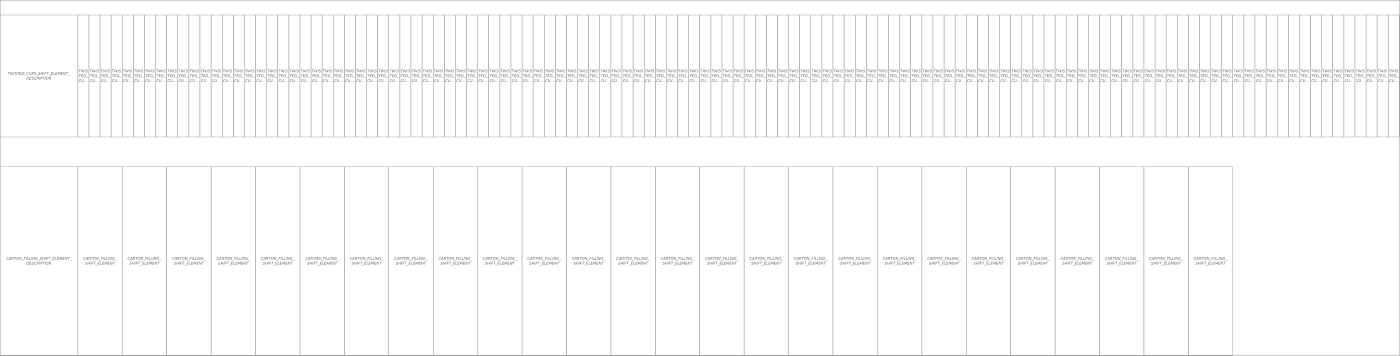
VISUALIZATION CUPS_PICK_AND_PLACE  // 3782x962
    Frame (210,40 30x330)
        shows TWISTED_CUPS_SHIFT_ELEMENT(index := 50)
    Frame (240,40 30x330)
        shows TWISTED_CUPS_SHIFT_ELEMENT(index := 51)
    Frame (270,40 30x330)
        shows TWISTED_CUPS_SHIFT_ELEMENT(index := 52)
    Frame (300,40 30x330)
        shows TWISTED_CUPS_SHIFT_ELEMENT(index := 53)
    Frame (330,40 30x330)
        shows TWISTED_CUPS_SHIFT_ELEMENT(index := 54)
    Frame (360,40 30x330)
        shows TWISTED_CUPS_SHIFT_ELEMENT(index := 55)
    Frame (390,40 30x330)
        shows TWISTED_CUPS_SHIFT_ELEMENT(index := 56)
    Frame (420,40 30x330)
        shows TWISTED_CUPS_SHIFT_ELEMENT(index := 57)
    Frame (450,40 30x330)
        shows TWISTED_CUPS_SHIFT_ELEMENT(index := 58)
    Frame (480,40 30x330)
        shows TWISTED_CUPS_SHIFT_ELEMENT(index := 59)
    Frame (510,40 30x330)
        shows TWISTED_CUPS_SHIFT_ELEMENT(index := 60)
    Frame (0,40 210x330)
        shows TWISTED_CUPS_SHIFT_ELEMENT_DESCRIPTION()
    Frame (540,40 30x330)
        shows TWISTED_CUPS_SHIFT_ELEMENT(index := 61)
    Frame (570,40 30x330)
        shows TWISTED_CUPS_SHIFT_ELEMENT(index := 62)
    Frame (600,40 30x330)
        shows TWISTED_CUPS_SHIFT_ELEMENT(index := 63)
    Frame (630,40 30x330)
        shows TWISTED_CUPS_SHIFT_ELEMENT(index := 64)
    Frame (660,40 30x330)
        shows TWISTED_CUPS_SHIFT_ELEMENT(index := 65)
    Frame (690,40 30x330)
        shows TWISTED_CUPS_SHIFT_ELEMENT(index := 66)
    Frame (720,40 30x330)
        shows TWISTED_CUPS_SHIFT_ELEMENT(index := 67)
    Frame (750,40 30x330)
        shows TWISTED_CUPS_SHIFT_ELEMENT(index := 68)
    Frame (780,40 30x330)
        shows TWISTED_CUPS_SHIFT_ELEMENT(index := 69)
    Frame (810,40 30x330)
        shows TWISTED_CUPS_SHIFT_ELEMENT(index := 70)
    Frame (840,40 30x330)
        shows TWISTED_CUPS_SHIFT_ELEMENT(index := 71)
    Frame (870,40 30x330)
        shows TWISTED_CUPS_SHIFT_ELEMENT(index := 72)
    Frame (900,40 30x330)
        shows TWISTED_CUPS_SHIFT_ELEMENT(index := 73)
    Frame (930,40 30x330)
        shows TWISTED_CUPS_SHIFT_ELEMENT(index := 74)
    Frame (960,40 30x330)
        shows TWISTED_CUPS_SHIFT_ELEMENT(index := 75)
    Frame (990,40 30x330)
        shows TWISTED_CUPS_SHIFT_ELEMENT(index := 76)
    Frame (1020,40 30x330)
        shows TWISTED_CUPS_SHIFT_ELEMENT(index := 77)
    Frame (1050,40 30x330)
        shows TWISTED_CUPS_SHIFT_ELEMENT(index := 78)
    Frame (1080,40 30x330)
        shows TWISTED_CUPS_SHIFT_ELEMENT(index := 79)
    Frame (1110,40 30x330)
        shows TWISTED_CUPS_SHIFT_ELEMENT(index := 80)
    Frame (1140,40 30x330)
        shows TWISTED_CUPS_SHIFT_ELEMENT(index := 81)
    Frame (1170,40 30x330)
        shows TWISTED_CUPS_SHIFT_ELEMENT(index := 82)
    Frame (1200,40 30x330)
        shows TWISTED_CUPS_SHIFT_ELEMENT(index := 83)
    Frame (1230,40 30x330)
        shows TWISTED_CUPS_SHIFT_ELEMENT(index := 84)
    Frame (1260,40 30x330)
        shows TWISTED_CUPS_SHIFT_ELEMENT(index := 85)
    Frame (1290,40 30x330)
        shows TWISTED_CUPS_SHIFT_ELEMENT(index := 86)
    Frame (1320,40 30x330)
        shows TWISTED_CUPS_SHIFT_ELEMENT(index := 87)
    Frame (1350,40 30x330)
        shows TWISTED_CUPS_SHIFT_ELEMENT(index := 88)
    Frame (1380,40 30x330)
        shows TWISTED_CUPS_SHIFT_ELEMENT(index := 89)
    Frame (1410,40 30x330)
        shows TWISTED_CUPS_SHIFT_ELEMENT(index := 90)
    Frame (1440,40 30x330)
        shows TWISTED_CUPS_SHIFT_ELEMENT(index := 91)
    Frame (1470,40 30x330)
        shows TWISTED_CUPS_SHIFT_ELEMENT(index := 92)
    Frame (1500,40 30x330)
        shows TWISTED_CUPS_SHIFT_ELEMENT(index := 93)
    Frame (1530,40 30x330)
        shows TWISTED_CUPS_SHIFT_ELEMENT(index := 94)
    Frame (1560,40 30x330)
        shows TWISTED_CUPS_SHIFT_ELEMENT(index := 95)
    Frame (1590,40 30x330)
        shows TWISTED_CUPS_SHIFT_ELEMENT(index := 96)
    Frame (1620,40 30x330)
        shows TWISTED_CUPS_SHIFT_ELEMENT(index := 97)
    Frame (1650,40 30x330)
        shows TWISTED_CUPS_SHIFT_ELEMENT(index := 98)
    Frame (1680,40 30x330)
        shows TWISTED_CUPS_SHIFT_ELEMENT(index := 99)
    Frame (1710,40 30x330)
        shows TWISTED_CUPS_SHIFT_ELEMENT(index := 100)
    Frame (1740,40 30x330)
        shows TWISTED_CUPS_SHIFT_ELEMENT(index := 101)
    Frame (1770,40 30x330)
        shows TWISTED_CUPS_SHIFT_ELEMENT(index := 102)
    Frame (1800,40 30x330)
        shows TWISTED_CUPS_SHIFT_ELEMENT(index := 103)
    Frame (1830,40 30x330)
        shows TWISTED_CUPS_SHIFT_ELEMENT(index := 104)
    Frame (1860,40 30x330)
        shows TWISTED_CUPS_SHIFT_ELEMENT(index := 105)
    Frame (1890,40 30x330)
        shows TWISTED_CUPS_SHIFT_ELEMENT(index := 106)
    Frame (1920,40 30x330)
        shows TWISTED_CUPS_SHIFT_ELEMENT(index := 107)
    Frame (1950,40 30x330)
        shows TWISTED_CUPS_SHIFT_ELEMENT(index := 108)
    Frame (1980,40 30x330)
        shows TWISTED_CUPS_SHIFT_ELEMENT(index := 109)
    Frame (2010,40 30x330)
        shows TWISTED_CUPS_SHIFT_ELEMENT(index := 110)
    Frame (2040,40 30x330)
        shows TWISTED_CUPS_SHIFT_ELEMENT(index := 111)
    Frame (2070,40 30x330)
        shows TWISTED_CUPS_SHIFT_ELEMENT(index := 112)
    Frame (2100,40 30x330)
        shows TWISTED_CUPS_SHIFT_ELEMENT(index := 113)
    Frame (2130,40 30x330)
        shows TWISTED_CUPS_SHIFT_ELEMENT(index := 114)
    Frame (2160,40 30x330)
        shows TWISTED_CUPS_SHIFT_ELEMENT(index := 115)
    Frame (2190,40 30x330)
        shows TWISTED_CUPS_SHIFT_ELEMENT(index := 116)
    Frame (2220,40 30x330)
        shows TWISTED_CUPS_SHIFT_ELEMENT(index := 117)
    Frame (2250,40 30x330)
        shows TWISTED_CUPS_SHIFT_ELEMENT(index := 118)
    Frame (2280,40 30x330)
        shows TWISTED_CUPS_SHIFT_ELEMENT(index := 119)
    Frame (2310,40 30x330)
        shows TWISTED_CUPS_SHIFT_ELEMENT(index := 120)
    Frame (0,450 210x510)
        shows CARTON_FILLING_SHIFT_ELEMENT_DESCRIPTION()
    Frame (2340,40 30x330)
        shows TWISTED_CUPS_SHIFT_ELEMENT(index := 121)
    Frame (2370,40 30x330)
        shows TWISTED_CUPS_SHIFT_ELEMENT(index := 122)
    Frame (2400,40 30x330)
        shows TWISTED_CUPS_SHIFT_ELEMENT(index := 123)
    Frame (2430,40 30x330)
        shows TWISTED_CUPS_SHIFT_ELEMENT(index := 124)
    Frame (2460,40 30x330)
        shows TWISTED_CUPS_SHIFT_ELEMENT(index := 125)
    Frame (2490,40 30x330)
        shows TWISTED_CUPS_SHIFT_ELEMENT(index := 126)
    Frame (2520,40 30x330)
        shows TWISTED_CUPS_SHIFT_ELEMENT(index := 127)
    Frame (2550,40 30x330)
        shows TWISTED_CUPS_SHIFT_ELEMENT(index := 128)
    Frame (2580,40 30x330)
        shows TWISTED_CUPS_SHIFT_ELEMENT(index := 129)
    Frame (2610,40 30x330)
        shows TWISTED_CUPS_SHIFT_ELEMENT(index := 130)
    Frame (2640,40 30x330)
        shows TWISTED_CUPS_SHIFT_ELEMENT(index := 131)
    Frame (2670,40 30x330)
        shows TWISTED_CUPS_SHIFT_ELEMENT(index := 132)
    Frame (2700,40 30x330)
        shows TWISTED_CUPS_SHIFT_ELEMENT(index := 133)
    Frame (2730,40 30x330)
        shows TWISTED_CUPS_SHIFT_ELEMENT(index := 134)
    Frame (2760,40 30x330)
        shows TWISTED_CUPS_SHIFT_ELEMENT(index := 135)
    Frame (2790,40 30x330)
        shows TWISTED_CUPS_SHIFT_ELEMENT(index := 136)
    Frame (2820,40 30x330)
        shows TWISTED_CUPS_SHIFT_ELEMENT(index := 137)
    Frame (2850,40 30x330)
        shows TWISTED_CUPS_SHIFT_ELEMENT(index := 138)
    Frame (2880,40 30x330)
        shows TWISTED_CUPS_SHIFT_ELEMENT(index := 139)
    Frame (2910,40 30x330)
        shows TWISTED_CUPS_SHIFT_ELEMENT(index := 140)
    Frame (2940,40 30x330)
        shows TWISTED_CUPS_SHIFT_ELEMENT(index := 141)
    Frame (2970,40 30x330)
        shows TWISTED_CUPS_SHIFT_ELEMENT(index := 142)
    Frame (3000,40 30x330)
        shows TWISTED_CUPS_SHIFT_ELEMENT(index := 143)
    Frame (3030,40 30x330)
        shows TWISTED_CUPS_SHIFT_ELEMENT(index := 144)
    Frame (3060,40 30x330)
        shows TWISTED_CUPS_SHIFT_ELEMENT(index := 145)
    Frame (3090,40 30x330)
        shows TWISTED_CUPS_SHIFT_ELEMENT(index := 146)
    Frame (3120,40 30x330)
        shows TWISTED_CUPS_SHIFT_ELEMENT(index := 147)
    Frame (3150,40 30x330)
        shows TWISTED_CUPS_SHIFT_ELEMENT(index := 148)
    Frame (3180,40 30x330)
        shows TWISTED_CUPS_SHIFT_ELEMENT(index := 149)
    Frame (3210,40 30x330)
        shows TWISTED_CUPS_SHIFT_ELEMENT(index := 150)
    Frame (3240,40 30x330)
        shows TWISTED_CUPS_SHIFT_ELEMENT(index := 151)
    Frame (3270,40 30x330)
        shows TWISTED_CUPS_SHIFT_ELEMENT(index := 152)
    Frame (3300,40 30x330)
        shows TWISTED_CUPS_SHIFT_ELEMENT(index := 153)
    Frame (3330,40 30x330)
        shows TWISTED_CUPS_SHIFT_ELEMENT(index := 154)
    Frame (3360,40 30x330)
        shows TWISTED_CUPS_SHIFT_ELEMENT(index := 155)
    Frame (3390,40 30x330)
        shows TWISTED_CUPS_SHIFT_ELEMENT(index := 156)
    Frame (3420,40 30x330)
        shows TWISTED_CUPS_SHIFT_ELEMENT(index := 157)
    Frame (3450,40 30x330)
        shows TWISTED_CUPS_SHIFT_ELEMENT(index := 158)
    Frame (3480,40 30x330)
        shows TWISTED_CUPS_SHIFT_ELEMENT(index := 159)
    Frame (3510,40 30x330)
        shows TWISTED_CUPS_SHIFT_ELEMENT(index := 160)
    Frame (3540,40 30x330)
        shows TWISTED_CUPS_SHIFT_ELEMENT(index := 161)
    Frame (3570,40 30x330)
        shows TWISTED_CUPS_SHIFT_ELEMENT(index := 162)
    Frame (3600,40 30x330)
        shows TWISTED_CUPS_SHIFT_ELEMENT(index := 163)
    Frame (3630,40 30x330)
        shows TWISTED_CUPS_SHIFT_ELEMENT(index := 164)
    Frame (3660,40 30x330)
        shows TWISTED_CUPS_SHIFT_ELEMENT(index := 165)
    Frame (3690,40 30x330)
        shows TWISTED_CUPS_SHIFT_ELEMENT(index := 166)
    Frame (3720,40 30x330)
        shows TWISTED_CUPS_SHIFT_ELEMENT(index := 167)
    Frame (3750,40 30x330)
        shows TWISTED_CUPS_SHIFT_ELEMENT(index := 168)
    Frame (210,450 120x510)
        shows CARTON_FILLING_SHIFT_ELEMENT(index := 135)
    Frame (330,450 120x510)
        shows CARTON_FILLING_SHIFT_ELEMENT(index := 134)
    Frame (450,450 120x510)
        shows CARTON_FILLING_SHIFT_ELEMENT(index := 133)
    Frame (570,450 120x510)
        shows CARTON_FILLING_SHIFT_ELEMENT(index := 132)
    Frame (690,450 120x510)
        shows CARTON_FILLING_SHIFT_ELEMENT(index := 131)
    Frame (810,450 120x510)
        shows CARTON_FILLING_SHIFT_ELEMENT(index := 130)
    Frame (930,450 120x510)
        shows CARTON_FILLING_SHIFT_ELEMENT(index := 129)
    Frame (1050,450 120x510)
        shows CARTON_FILLING_SHIFT_ELEMENT(index := 128)
    Frame (1170,450 120x510)
        shows CARTON_FILLING_SHIFT_ELEMENT(index := 127)
    Frame (1290,450 120x510)
        shows CARTON_FILLING_SHIFT_ELEMENT(index := 126)
    Frame (1410,450 120x510)
        shows CARTON_FILLING_SHIFT_ELEMENT(index := 125)
    Frame (1530,450 120x510)
        shows CARTON_FILLING_SHIFT_ELEMENT(index := 124)
    Frame (1650,450 120x510)
        shows CARTON_FILLING_SHIFT_ELEMENT(index := 123)
    Frame (1770,450 120x510)
        shows CARTON_FILLING_SHIFT_ELEMENT(index := 122)
    Frame (1890,450 120x510)
        shows CARTON_FILLING_SHIFT_ELEMENT(index := 121)
    Frame (2010,450 120x510)
        shows CARTON_FILLING_SHIFT_ELEMENT(index := 120)
    Frame (2130,450 120x510)
        shows CARTON_FILLING_SHIFT_ELEMENT(index := 119)
    Frame (2250,450 120x510)
        shows CARTON_FILLING_SHIFT_ELEMENT(index := 118)
    Frame (2370,450 120x510)
        shows CARTON_FILLING_SHIFT_ELEMENT(index := 117)
    Frame (2490,450 120x510)
        shows CARTON_FILLING_SHIFT_ELEMENT(index := 116)
    Frame (2610,450 120x510)
        shows CARTON_FILLING_SHIFT_ELEMENT(index := 115)
    Frame (2730,450 120x510)
        shows CARTON_FILLING_SHIFT_ELEMENT(index := 114)
    Frame (2850,450 120x510)
        shows CARTON_FILLING_SHIFT_ELEMENT(index := 113)
    Frame (2970,450 120x510)
        shows CARTON_FILLING_SHIFT_ELEMENT(index := 112)
    Frame (3090,450 120x510)
        shows CARTON_FILLING_SHIFT_ELEMENT(index := 111)
    Frame (3210,450 120x510)
        shows CARTON_FILLING_SHIFT_ELEMENT(index := 110)
END_VISUALIZATION

(* stored: Version 1.1.0.1, ProductVersion 3.1.4024.3
   Visu CUPS_PICK_AND_PLACE: Id {5ce4712c-5c8d-44a8-b902-4fba432da6c6} *)
